FUNCTION_BLOCK ButtonController
VAR_INPUT
	StartButton: BOOL;
	ResetButton: BOOL;
	StopButton: BOOL;
	EmgStopButton: BOOL;
END_VAR
VAR_OUTPUT
	StartLight: BOOL;
	ResetLight: BOOL;
	StopLight: BOOL;
END_VAR
VAR
	tBlink: TON;
END_VAR

// Blinking logic
tBlink(IN := NOT tBlink.Q, PT := T#1000MS);
GVL.BlinkBit := tBlink.ET > T#500MS;
// -------------
// Memory Bit For SystemON (when true the system is ready to run)
IF GVL.isStopON THEN
	IF NOT GVL.isEmgStopON AND StartButton THEN
		GVL.isSystemON := TRUE;
	END_IF;
END_IF;
IF GVL.isResetON THEN
	IF NOT GVL.isEmgStopON AND StartButton AND NOT GVL.isStopON THEN
		GVL.isSystemON := TRUE;
	END_IF;
END_IF;
IF GVL.isEmgStopON OR NOT StopButton THEN
	GVL.isSystemON := FALSE;
END_IF;
// -------------
// Memory bit for IsEmgStopON - Set/Reset
IF NOT EmgStopButton THEN
	GVL.isEmgStopON := TRUE;
END_IF;
IF EmgStopButton THEN
	GVL.isEmgStopON := FALSE;
END_IF;
// -------------
// Memory bit for IsResetON - Set/Reset
IF ResetButton AND NOT GVL.isEmgStopON AND NOT GVL.isStopON THEN
	GVL.isResetON := TRUE;
END_IF;
IF StartButton THEN
	GVL.isResetON := FALSE;
END_IF;
// -------------
// Memory bit for IsStopON - Set/Reset
IF NOT StopButton AND NOT GVL.isEmgStopON THEN
	GVL.isStopON := TRUE;
END_IF;
IF GVL.isSystemON OR GVL.wasEmgBtnPressed THEN
	GVL.isStopON := FALSE;
END_IF;
// -------------
// Memory bit for wasEmgBtnPressed - Set/Reset
IF NOT EmgStopButton THEN
	GVL.wasEmgBtnPressed := TRUE;
	GVL.isResetON := FALSE;
END_IF;
IF GVL.isSystemON THEN
	GVL.wasEmgBtnPressed := FALSE;
END_IF;
// ------------- OUTPUTS --------------
StartLight := GVL.isSystemON OR ((GVL.isResetON OR (NOT GVL.isResetON AND GVL.isStopON)) AND NOT GVL.isEmgStopON AND NOT GVL.isSystemON AND GVL.BlinkBit);
ResetLight := (GVL.isResetON OR (NOT GVL.isResetON AND GVL.BlinkBit)) AND NOT GVL.isEmgStopON AND NOT GVL.isStopON AND NOT GVL.isSystemON;
StopLight := (GVL.isEmgStopON OR GVL.isStopON) AND NOT GVL.isSystemON;

END_FUNCTION_BLOCK

(* stored: Version 1.1.0.1, ProductVersion 3.1.4024.12
   POU ButtonController: Id {80405ffb-ef53-44cb-b1a4-4e4b684fba13}, SpecialFunc None *)
